// TIA Portal V19 export
TYPE "Positioning_EPOS_Machine_Par"
// stored: Access Published
   STRUCT
      PosTolerance { S7_SetPoint := 'True'} : LReal;   // mm
      DelayInPosition : Time;
      Man_Vel { S7_SetPoint := 'True'} : LReal;   // Override 0-100% delle speed
      Man_Acc : LReal;
      Man_Dec : LReal;
   END_STRUCT;
END_TYPE
